(* CODESYS project TP2_INF_IND_RENAN_JULIA.project

Project tree, tasks and I/O mapping:
  Device : CODESYS Control Win V3, 3S - Smart Software Solutions GmbH, order no. 305021, version 3.5.11.40
    application Application
      libraries: Standard, * (System)
      task MainTask (cyclic, interval t#20ms, priority 1) calls Main
      task Simulacao (cyclic, interval t#20ms, priority 1) calls SimulacaoProcesso
      program Main [ST]
      Symbols
      function block AlarmLogic [ST]
      program SimulacaoProcesso [ST]
*)

// Device/Application/Main
PROGRAM Main
VAR_INPUT
    CMD_INICIAR_CARREGAMENTO: BOOL;
    CMD_INICIAR_DESCARREGAMENTO: BOOL;
    CAMINHAO_POSICIONADO: BOOL;
    CAPACIDADE_CAMINHAO: REAL;
    PESO_SILO1: REAL;
    PESO_SILO2: REAL;
    Modo_Automatico_Carregamento: BOOL;
    Modo_Automatico_Descarregamento: BOOL;
    CMD_MANUAL_VENTILACAO_SILO1: BOOL;
    CMD_MANUAL_VENTILACAO_SILO2: BOOL;
    CMD_MANUAL_ALIMENTADOR_MOEGA1_ON: BOOL;
    CMD_MANUAL_ALIMENTADOR_MOEGA2_ON: BOOL;
    CMD_MANUAL_TRANSPORTADOR_ENTRADA_ON: BOOL;
    CMD_MANUAL_TRANSPORTADOR_SAIDA_ON: BOOL;
    CMD_MANUAL_MOEGA_PESAGEM_ON: BOOL;
    CMD_MANUAL_ALIMENTADOR_SAIDA_ON: BOOL;
    CMD_MANUAL_DESVIADOR_MANGUEIRA: INT;
END_VAR

VAR_OUTPUT
    VENTILACAO_SILO1: BOOL := FALSE;
    VENTILACAO_SILO2: BOOL := FALSE;
    ALIMENTADOR_MOEGA1_ON: BOOL := FALSE;
    ALIMENTADOR_MOEGA2_ON: BOOL := FALSE;
    TRANSPORTADOR_SAIDA_ON: BOOL := FALSE;
    MOEGA_PESAGEM_ON: BOOL := FALSE;
    TRANSPORTADOR_ENTRADA_ON: BOOL := FALSE;
    DESVIADOR_MANGUEIRA: INT :=1;
END_VAR

VAR
	alarmLogic: AlarmLogic;
    NIVEL_BAIXO_SILO1: BOOL;
    NIVEL_BAIXO_SILO2: BOOL;
    NIVEL_ALTO_SILO1: BOOL;
    NIVEL_ALTO_SILO2: BOOL;
    PESO_MOEGA: REAL;
    TaxaTransferenciaCarregamento: REAL := 50.0;
    TaxaTransferenciaDescarregamento: REAL := 100.0;
    ALARME_CARREGAMENTO: BOOL;
    ALARME_DESCARREGAMENTO: BOOL;
    INICIAR_CARREGAMENTO: BOOL;
    INICIAR_DESCARREGAMENTO: BOOL;
    inicio_carregamento: TIME;
    inicio_descarregamento: TIME;
    SiloSelecionado: INT;
    VAGAO_POSICIONADO: BOOL;
    CAPACIDADE_VAGAO: REAL := 1000.0;
    VAGAO_CAPACIDADE_RESTANTE: REAL := 0.0;
    VAGAO_POSICIONADO_ANTERIOR: BOOL := FALSE;
    lastUpdateTime: TIME;
    elapsedTime: REAL;
    CAMINHAO_CHEIO: BOOL;
    equipmentOffTime: TIME;
    VAGAO_CHEIO: BOOL;
    CapacidadeDisponivelSilo1: REAL;
    CapacidadeDisponivelSilo2: REAL;
    CapacidadeTotalDisponivel: REAL;
    CapacidadeDescarregamento: REAL := 1000.0;
    CAMINHAO_POSICIONADO_ANTERIOR: BOOL := FALSE;
	ALARME_TRANSPORTADOR_ENTRADA_VAZIO: BOOL;
	ALARME_ALIMENTADOR_MOEGA_VAZIO: BOOL;
	ALARME_MOEGA_PESAGEM: BOOL;
	ALIMENTADOR_SAIDA_ON: BOOL;
	ALARME_TRANSPORTADOR_SAIDA_VAZIO: BOOL;
	ALARME_ALIMENTADOR_SAIDA: BOOL;
	ALARME_TRANSPORTADOR_SAIDA_ALIMENTADOR: BOOL;
	TRANSPORTADOR_ENTRADA_VAZIO_TIMER: TIME;
    TRANSPORTADOR_ENTRADA_VAZIO: BOOL := FALSE;
    
    PESO_TRANSPORTADOR_ENTRADA: REAL;
	ALARME_TRANSPORTADOR_ENTRADA_CHEIO: BOOL;
	TIMER_ALIMENTADOR_MOEGA1_VAZIO: TIME;
    ALARME_ALIMENTADOR_MOEGA1_VAZIO: BOOL := FALSE;
    ALARME_ALIMENTADOR_MOEGA1_CHEIO: BOOL := FALSE;
    PESO_ALIMENTADOR_MOEGA1: REAL; 

    TIMER_ALIMENTADOR_MOEGA2_VAZIO: TIME;
    ALARME_ALIMENTADOR_MOEGA2_VAZIO: BOOL := FALSE;
    ALARME_ALIMENTADOR_MOEGA2_CHEIO: BOOL := FALSE;
    PESO_ALIMENTADOR_MOEGA2: REAL;
	TIMER_TRANSPORTADOR_SAIDA_VAZIO: TIME;
	TIMER_TRANSPORTADOR_ENTRADA_VAZIO: TIME;
	PermiteMudancaModoCarregamento: BOOL := FALSE;
	PermiteMudancaModoDescarregamento: BOOL:= FALSE;
	VAGAO_FORA: BOOL;
	AUTORIZA_CARREGAMENTO: BOOL;
	ALARMES_DESLIGADOS: BOOL;
	DESCARREGAMENTO_EM_ANDAMENTO: BOOL;
END_VAR

alarmLogic.CURRENT_TIME := TIME();

// Configurar entradas do Function Block
alarmLogic.MOEGA_PESAGEM_ON := MOEGA_PESAGEM_ON;
alarmLogic.PESO_MOEGA := PESO_MOEGA;
alarmLogic.TRANSPORTADOR_SAIDA_ON := TRANSPORTADOR_SAIDA_ON;
alarmLogic.ALIMENTADOR_SAIDA_ON := ALIMENTADOR_SAIDA_ON;
alarmLogic.TRANSPORTADOR_ENTRADA_ON := TRANSPORTADOR_ENTRADA_ON;
alarmLogic.PESO_TRANSPORTADOR_ENTRADA := PESO_TRANSPORTADOR_ENTRADA;
alarmLogic.ALIMENTADOR_MOEGA1_ON := ALIMENTADOR_MOEGA1_ON;
alarmLogic.PESO_ALIMENTADOR_MOEGA1 := PESO_ALIMENTADOR_MOEGA1;
alarmLogic.ALIMENTADOR_MOEGA2_ON := ALIMENTADOR_MOEGA2_ON;
alarmLogic.PESO_ALIMENTADOR_MOEGA2 := PESO_ALIMENTADOR_MOEGA2;
alarmLogic.CAMINHAO_POSICIONADO := CAMINHAO_POSICIONADO;

// Chamar o Function Block
alarmLogic();

// Ler saídas do Function Block
ALARME_MOEGA_PESAGEM := alarmLogic.ALARME_MOEGA_PESAGEM;
ALARME_TRANSPORTADOR_SAIDA_VAZIO := alarmLogic.ALARME_TRANSPORTADOR_SAIDA_VAZIO;
ALARME_TRANSPORTADOR_SAIDA_ALIMENTADOR := alarmLogic.ALARME_TRANSPORTADOR_SAIDA_ALIMENTADOR;
ALARME_TRANSPORTADOR_ENTRADA_VAZIO := alarmLogic.ALARME_TRANSPORTADOR_ENTRADA_VAZIO;
ALARME_TRANSPORTADOR_ENTRADA_CHEIO := alarmLogic.ALARME_TRANSPORTADOR_ENTRADA_CHEIO;
ALARME_ALIMENTADOR_MOEGA1_VAZIO := alarmLogic.ALARME_ALIMENTADOR_MOEGA1_VAZIO;
ALARME_ALIMENTADOR_MOEGA1_CHEIO := alarmLogic.ALARME_ALIMENTADOR_MOEGA1_CHEIO;
ALARME_ALIMENTADOR_MOEGA2_VAZIO := alarmLogic.ALARME_ALIMENTADOR_MOEGA2_VAZIO;
ALARME_ALIMENTADOR_MOEGA2_CHEIO := alarmLogic.ALARME_ALIMENTADOR_MOEGA2_CHEIO;
ALARME_ALIMENTADOR_SAIDA := alarmLogic.ALARME_ALIMENTADOR_SAIDA;
ALARMES_DESLIGADOS    := alarmLogic.ALARMES_DESLIGADOS;

IF PESO_SILO1 <= 100 THEN
    NIVEL_BAIXO_SILO1 := TRUE;
ELSE
    NIVEL_BAIXO_SILO1 := FALSE;    
END_IF

IF PESO_SILO2 <= 100 THEN
    NIVEL_BAIXO_SILO2 := TRUE;
ELSE
    NIVEL_BAIXO_SILO2 := FALSE;    
END_IF

IF PESO_SILO1 >= 2400 THEN
    NIVEL_ALTO_SILO1 := TRUE;
ELSE
    NIVEL_ALTO_SILO1 := FALSE;    
END_IF

IF PESO_SILO2 >= 2400 THEN
    NIVEL_ALTO_SILO2 := TRUE;
ELSE 
    NIVEL_ALTO_SILO2 := FALSE;    
END_IF

IF TRANSPORTADOR_ENTRADA_ON AND (NOT VAGAO_POSICIONADO) THEN
	VAGAO_FORA := TRUE;
ELSE
    VAGAO_FORA := FALSE;	
END_IF

elapsedTime := TIME_TO_REAL(TIME() - lastUpdateTime) / 1000.0;
lastUpdateTime := TIME();

IF VAGAO_POSICIONADO AND NOT VAGAO_POSICIONADO_ANTERIOR THEN
    VAGAO_CAPACIDADE_RESTANTE := CAPACIDADE_VAGAO;
    VAGAO_POSICIONADO_ANTERIOR := TRUE;
    VAGAO_CHEIO := FALSE;
ELSIF NOT VAGAO_POSICIONADO THEN
    VAGAO_POSICIONADO_ANTERIOR := FALSE;
END_IF

IF CAMINHAO_POSICIONADO AND NOT CAMINHAO_POSICIONADO_ANTERIOR THEN
    CAMINHAO_POSICIONADO_ANTERIOR := TRUE;
    CAMINHAO_CHEIO := FALSE;
    AUTORIZA_CARREGAMENTO := TRUE; // Autoriza carregamento quando caminhão é reposicionado
ELSIF NOT CAMINHAO_POSICIONADO THEN
    CAMINHAO_POSICIONADO_ANTERIOR := FALSE;
    AUTORIZA_CARREGAMENTO := FALSE; // Reseta a autorização quando caminhão não está mais posicionado
END_IF

// Carregamento
IF Modo_Automatico_Carregamento THEN
    IF NOT INICIAR_CARREGAMENTO AND CMD_INICIAR_CARREGAMENTO AND AUTORIZA_CARREGAMENTO THEN
        IF CAMINHAO_POSICIONADO AND (CAPACIDADE_CAMINHAO >= 200 AND CAPACIDADE_CAMINHAO <= 800 AND (REAL_TO_INT(CAPACIDADE_CAMINHAO) MOD 50 = 0)) THEN
            IF ((PESO_SILO1 - 100) + (PESO_SILO2 - 100) >= CAPACIDADE_CAMINHAO) AND (NOT CAMINHAO_CHEIO) THEN
                INICIAR_CARREGAMENTO := TRUE;
                inicio_carregamento := TIME();
                ALARME_CARREGAMENTO := FALSE;

                IF PESO_SILO1 >= PESO_SILO2 THEN
                    SiloSelecionado := 1;
                ELSE
                    SiloSelecionado := 2;
                END_IF;
            ELSE
                ALARME_CARREGAMENTO := TRUE;
            END_IF
        ELSE
            ALARME_CARREGAMENTO := TRUE;
        END_IF
    END_IF

    IF INICIAR_CARREGAMENTO THEN
        IF (PESO_SILO1 >= 100 OR PESO_SILO2 >= 100) THEN
            TRANSPORTADOR_SAIDA_ON := TRUE;
            MOEGA_PESAGEM_ON := TRUE;
            ALIMENTADOR_SAIDA_ON := TRUE;

            IF PESO_MOEGA < CAPACIDADE_CAMINHAO THEN
                PESO_MOEGA := PESO_MOEGA + TaxaTransferenciaCarregamento * elapsedTime;
                IF SiloSelecionado = 1 THEN
                    IF NOT NIVEL_BAIXO_SILO1 THEN
                        VENTILACAO_SILO1 := TRUE; 
                        PESO_SILO1 := PESO_SILO1 - TaxaTransferenciaCarregamento * elapsedTime;
                        ALIMENTADOR_MOEGA1_ON := TRUE;
                        PESO_ALIMENTADOR_MOEGA1 := 1;
                        PESO_ALIMENTADOR_MOEGA2 := 0;
                        VENTILACAO_SILO2 := FALSE;
                        ALIMENTADOR_MOEGA2_ON := FALSE;
                    ELSE
                        SiloSelecionado := 2;
                        VENTILACAO_SILO1 := FALSE;
                        VENTILACAO_SILO2 := TRUE;
                    END_IF;
                ELSIF SiloSelecionado = 2 THEN
                    IF NOT NIVEL_BAIXO_SILO2 THEN
                        VENTILACAO_SILO2 := TRUE;
                        PESO_SILO2 := PESO_SILO2 - TaxaTransferenciaCarregamento * elapsedTime;
                        ALIMENTADOR_MOEGA2_ON := TRUE;
                        PESO_ALIMENTADOR_MOEGA1 := 0;
                        PESO_ALIMENTADOR_MOEGA2 := 1;
                        VENTILACAO_SILO1 := FALSE;
                        ALIMENTADOR_MOEGA1_ON := FALSE;
                    ELSE
                        SiloSelecionado := 1;
                        VENTILACAO_SILO1 := TRUE;
                        VENTILACAO_SILO2 := FALSE;
                    END_IF;
                END_IF;
            END_IF
        ELSE
            ALARME_CARREGAMENTO := TRUE;
            INICIAR_CARREGAMENTO := FALSE;
        END_IF;

        IF PESO_MOEGA >= CAPACIDADE_CAMINHAO OR ALARME_ALIMENTADOR_SAIDA THEN
            CAMINHAO_CHEIO := TRUE;
            INICIAR_CARREGAMENTO := FALSE;
            equipmentOffTime := TIME();
            AUTORIZA_CARREGAMENTO := FALSE; // Reseta a autorização após o carregamento ser concluído
        END_IF
    END_IF

    IF CAMINHAO_CHEIO THEN
        ALIMENTADOR_MOEGA1_ON := FALSE;
        PESO_ALIMENTADOR_MOEGA1 := 0;
        ALIMENTADOR_MOEGA2_ON := FALSE;
        PESO_ALIMENTADOR_MOEGA2 := 0;
        IF (TIME() - equipmentOffTime >= T#1S) THEN
            MOEGA_PESAGEM_ON := FALSE;
            PESO_MOEGA := 0;
        END_IF
        IF (TIME() - equipmentOffTime >= T#2S) THEN
            TRANSPORTADOR_SAIDA_ON := FALSE;
        END_IF
        IF (TIME() - equipmentOffTime >= T#3S) THEN
            ALIMENTADOR_SAIDA_ON := FALSE;
        END_IF
        IF (TIME() - equipmentOffTime >= T#5S) THEN
            VENTILACAO_SILO1 := FALSE;
            VENTILACAO_SILO2 := FALSE;
            CAMINHAO_CHEIO := FALSE;
        END_IF
    END_IF
END_IF

// Descarregamento
IF Modo_Automatico_Descarregamento THEN
    CapacidadeDisponivelSilo1 := 2400.0 - PESO_SILO1;
    CapacidadeDisponivelSilo2 := 2400.0 - PESO_SILO2;
    CapacidadeTotalDisponivel := CapacidadeDisponivelSilo1 + CapacidadeDisponivelSilo2;

    IF NOT INICIAR_DESCARREGAMENTO AND CMD_INICIAR_DESCARREGAMENTO THEN
        IF VAGAO_POSICIONADO AND (CapacidadeTotalDisponivel >= CapacidadeDescarregamento) AND (NOT VAGAO_CHEIO OR NOT VAGAO_FORA) AND NOT (NIVEL_ALTO_SILO1 AND NIVEL_ALTO_SILO2) THEN
            IF NOT ALARME_DESCARREGAMENTO THEN
                INICIAR_DESCARREGAMENTO := TRUE;
                inicio_descarregamento := TIME();
                ALARME_DESCARREGAMENTO := FALSE;

                IF (PESO_SILO1 < PESO_SILO2) AND (NOT NIVEL_ALTO_SILO1) THEN
                    DESVIADOR_MANGUEIRA := 1;
                    VENTILACAO_SILO1 := TRUE;
                    VENTILACAO_SILO2 := FALSE;
                ELSIF (PESO_SILO2 < PESO_SILO1) AND (NOT NIVEL_ALTO_SILO2) THEN
                    DESVIADOR_MANGUEIRA := 2;
                    VENTILACAO_SILO2 := TRUE;
                    VENTILACAO_SILO1 := FALSE;
                ELSIF (PESO_SILO1 = PESO_SILO2) THEN
                    IF NOT INICIAR_DESCARREGAMENTO THEN
                        IF DESVIADOR_MANGUEIRA = 1 THEN
                            SiloSelecionado := 1;
                            DESVIADOR_MANGUEIRA := 1;
                            VENTILACAO_SILO1 := TRUE;
                            VENTILACAO_SILO2 := FALSE;
                        ELSE
                            SiloSelecionado := 2;
                            DESVIADOR_MANGUEIRA := 2;
                            VENTILACAO_SILO2 := TRUE;
                            VENTILACAO_SILO1 := FALSE;
                        END_IF
                    END_IF
                END_IF
            END_IF
        ELSE
            ALARME_DESCARREGAMENTO := TRUE;
        END_IF
    END_IF

    IF INICIAR_DESCARREGAMENTO THEN
        TRANSPORTADOR_ENTRADA_ON := TRUE;
        
        PESO_TRANSPORTADOR_ENTRADA := 1;
        IF VAGAO_CAPACIDADE_RESTANTE > 0 THEN
            IF (NOT NIVEL_ALTO_SILO1) AND (DESVIADOR_MANGUEIRA = 1) THEN
                PESO_SILO1 := PESO_SILO1 + TaxaTransferenciaDescarregamento * elapsedTime;
                VAGAO_CAPACIDADE_RESTANTE := VAGAO_CAPACIDADE_RESTANTE - TaxaTransferenciaDescarregamento * elapsedTime;
                VENTILACAO_SILO1 := TRUE;
                VENTILACAO_SILO2 := FALSE;
                IF NIVEL_ALTO_SILO1 THEN
                    DESVIADOR_MANGUEIRA := 2;
                    VENTILACAO_SILO1 := FALSE;
                    VENTILACAO_SILO2 := TRUE;
                END_IF
            ELSE
                IF (NOT NIVEL_ALTO_SILO2) THEN
                    PESO_SILO2 := PESO_SILO2 + TaxaTransferenciaDescarregamento * elapsedTime;
                    VAGAO_CAPACIDADE_RESTANTE := VAGAO_CAPACIDADE_RESTANTE - TaxaTransferenciaDescarregamento * elapsedTime;
                    VENTILACAO_SILO2 := TRUE;
                    VENTILACAO_SILO1 := FALSE;
                    DESVIADOR_MANGUEIRA := 2;
                    
                END_IF
                IF NIVEL_ALTO_SILO2 THEN
                    DESVIADOR_MANGUEIRA := 1;
                    VENTILACAO_SILO2 := FALSE;
                    VENTILACAO_SILO1 := TRUE;
                END_IF
            END_IF

            IF VAGAO_CAPACIDADE_RESTANTE <= 0 OR VAGAO_FORA THEN
                VAGAO_CHEIO := TRUE;
                INICIAR_DESCARREGAMENTO := FALSE;
                equipmentOffTime := TIME();
            END_IF
        END_IF
    END_IF

    IF VAGAO_CHEIO THEN
        IF (TIME() - equipmentOffTime >= T#2S) THEN
            TRANSPORTADOR_ENTRADA_ON := FALSE;
            PESO_TRANSPORTADOR_ENTRADA := 0;
        END_IF
        IF (TIME() - equipmentOffTime >= T#5S) THEN
            VENTILACAO_SILO1 := FALSE;
            VENTILACAO_SILO2 := FALSE;
        END_IF
    END_IF

    // Redefinir alarme quando houver capacidade
    IF CapacidadeTotalDisponivel >= CapacidadeDescarregamento THEN
        ALARME_DESCARREGAMENTO := FALSE;
    END_IF
END_IF


IF NOT Modo_Automatico_Carregamento THEN
    IF ALARMES_DESLIGADOS THEN
        VENTILACAO_SILO1 := CMD_MANUAL_VENTILACAO_SILO1;
        VENTILACAO_SILO2 := CMD_MANUAL_VENTILACAO_SILO2;
        ALIMENTADOR_MOEGA1_ON := CMD_MANUAL_ALIMENTADOR_MOEGA1_ON;
        ALIMENTADOR_MOEGA2_ON := CMD_MANUAL_ALIMENTADOR_MOEGA2_ON;
        TRANSPORTADOR_SAIDA_ON := CMD_MANUAL_TRANSPORTADOR_SAIDA_ON;
        MOEGA_PESAGEM_ON := CMD_MANUAL_MOEGA_PESAGEM_ON;
    END_IF
END_IF

IF NOT Modo_Automatico_Descarregamento THEN
    IF ALARMES_DESLIGADOS THEN
        VENTILACAO_SILO1 := CMD_MANUAL_VENTILACAO_SILO1;
        VENTILACAO_SILO2 := CMD_MANUAL_VENTILACAO_SILO2;
        DESVIADOR_MANGUEIRA := CMD_MANUAL_DESVIADOR_MANGUEIRA;
        TRANSPORTADOR_ENTRADA_ON := CMD_MANUAL_TRANSPORTADOR_ENTRADA_ON;
    END_IF
END_IF

END_PROGRAM

// Device/Application/AlarmLogic
FUNCTION_BLOCK AlarmLogic
VAR_INPUT
    MOEGA_PESAGEM_ON: BOOL;
    PESO_MOEGA: REAL;
    TRANSPORTADOR_SAIDA_ON: BOOL;
    ALIMENTADOR_SAIDA_ON: BOOL;
    TRANSPORTADOR_ENTRADA_ON: BOOL;
    PESO_TRANSPORTADOR_ENTRADA: REAL;
    ALIMENTADOR_MOEGA1_ON: BOOL;
    PESO_ALIMENTADOR_MOEGA1: REAL;
    ALIMENTADOR_MOEGA2_ON: BOOL;
    PESO_ALIMENTADOR_MOEGA2: REAL;
	CURRENT_TIME: TIME;
	CAMINHAO_POSICIONADO :BOOL;
END_VAR

VAR_OUTPUT
    ALARME_MOEGA_PESAGEM: BOOL;
    ALARME_TRANSPORTADOR_SAIDA_VAZIO: BOOL;
    ALARME_TRANSPORTADOR_SAIDA_ALIMENTADOR: BOOL;
    ALARME_TRANSPORTADOR_ENTRADA_VAZIO: BOOL;
    ALARME_TRANSPORTADOR_ENTRADA_CHEIO: BOOL;
    ALARME_ALIMENTADOR_MOEGA1_VAZIO: BOOL;
    ALARME_ALIMENTADOR_MOEGA1_CHEIO: BOOL;
    ALARME_ALIMENTADOR_MOEGA2_VAZIO: BOOL;
    ALARME_ALIMENTADOR_MOEGA2_CHEIO: BOOL;
	ALARME_ALIMENTADOR_SAIDA : BOOL;
	ALARMES_DESLIGADOS: BOOL;
END_VAR

VAR
    TIMER_TRANSPORTADOR_SAIDA_VAZIO: TIME;
    TIMER_TRANSPORTADOR_ENTRADA_VAZIO: TIME;
    TIMER_ALIMENTADOR_MOEGA1_VAZIO: TIME;
    TIMER_ALIMENTADOR_MOEGA2_VAZIO: TIME;

	
END_VAR

// Alarme para moega de pesagem com peso diferente de zero e transportador de saída desligado
IF (MOEGA_PESAGEM_ON AND (PESO_MOEGA > 0)) AND NOT TRANSPORTADOR_SAIDA_ON THEN
    ALARME_MOEGA_PESAGEM := TRUE;
ELSE
    ALARME_MOEGA_PESAGEM := FALSE;
END_IF

// Alarme para transportador de saída vazio por mais de 5 segundos
IF TRANSPORTADOR_SAIDA_ON AND (PESO_MOEGA <= 0) THEN
    IF (CURRENT_TIME - TIMER_TRANSPORTADOR_SAIDA_VAZIO >= T#5S) THEN
        ALARME_TRANSPORTADOR_SAIDA_VAZIO := TRUE;
    END_IF
ELSE
    ALARME_TRANSPORTADOR_SAIDA_VAZIO := FALSE;
    TIMER_TRANSPORTADOR_SAIDA_VAZIO := CURRENT_TIME;
END_IF

// Alarme para transportador de saída ligado e alimentador de saída desligado
IF TRANSPORTADOR_SAIDA_ON AND NOT ALIMENTADOR_SAIDA_ON THEN
    ALARME_TRANSPORTADOR_SAIDA_ALIMENTADOR := TRUE;
ELSE
    ALARME_TRANSPORTADOR_SAIDA_ALIMENTADOR := FALSE;
END_IF

// Alarme para transportador de entrada vazio por mais de 5 segundos
IF TRANSPORTADOR_ENTRADA_ON AND (PESO_TRANSPORTADOR_ENTRADA <= 0) THEN
    IF (CURRENT_TIME - TIMER_TRANSPORTADOR_ENTRADA_VAZIO >= T#5S) THEN
        ALARME_TRANSPORTADOR_ENTRADA_VAZIO := TRUE;
    END_IF
ELSE
    ALARME_TRANSPORTADOR_ENTRADA_VAZIO := FALSE;
    TIMER_TRANSPORTADOR_ENTRADA_VAZIO := CURRENT_TIME;
END_IF

// Alarme para transportador de entrada quando há material dentro de si
IF TRANSPORTADOR_ENTRADA_ON AND (PESO_TRANSPORTADOR_ENTRADA > 0) THEN
    ALARME_TRANSPORTADOR_ENTRADA_CHEIO := TRUE;
ELSE
    ALARME_TRANSPORTADOR_ENTRADA_CHEIO := FALSE;
END_IF

// Alarme para Alimentador da Moega 1 vazio por mais de 5 segundos
IF ALIMENTADOR_MOEGA1_ON AND (PESO_ALIMENTADOR_MOEGA1 <= 0) THEN
    IF (CURRENT_TIME - TIMER_ALIMENTADOR_MOEGA1_VAZIO >= T#5S) THEN
        ALARME_ALIMENTADOR_MOEGA1_VAZIO := TRUE;
    END_IF
ELSE
    ALARME_ALIMENTADOR_MOEGA1_VAZIO := FALSE;
    TIMER_ALIMENTADOR_MOEGA1_VAZIO := CURRENT_TIME;
END_IF

// Alarme para Alimentador da Moega 1 quando há grãos no alimentador
IF ALIMENTADOR_MOEGA1_ON AND (PESO_ALIMENTADOR_MOEGA1 > 0) THEN
    ALARME_ALIMENTADOR_MOEGA1_CHEIO := TRUE;
ELSE
    ALARME_ALIMENTADOR_MOEGA1_CHEIO := FALSE;
END_IF

// Alarme para Alimentador da Moega 2 vazio por mais de 5 segundos
IF ALIMENTADOR_MOEGA2_ON AND (PESO_ALIMENTADOR_MOEGA2 <= 0) THEN
    IF (CURRENT_TIME - TIMER_ALIMENTADOR_MOEGA2_VAZIO >= T#5S) THEN
        ALARME_ALIMENTADOR_MOEGA2_VAZIO := TRUE;
    END_IF
ELSE
    ALARME_ALIMENTADOR_MOEGA2_VAZIO := FALSE;
    TIMER_ALIMENTADOR_MOEGA2_VAZIO := CURRENT_TIME;
END_IF

// Alarme para Alimentador da Moega 2 quando há grãos no alimentador
IF ALIMENTADOR_MOEGA2_ON AND (PESO_ALIMENTADOR_MOEGA2 > 0) THEN
    ALARME_ALIMENTADOR_MOEGA2_CHEIO := TRUE;
ELSE
    ALARME_ALIMENTADOR_MOEGA2_CHEIO := FALSE;
END_IF

IF ALIMENTADOR_SAIDA_ON AND (NOT CAMINHAO_POSICIONADO) THEN
	ALARME_ALIMENTADOR_SAIDA := TRUE;
ELSE
    ALARME_ALIMENTADOR_SAIDA := FALSE;	
END_IF


IF NOT ALARME_ALIMENTADOR_SAIDA AND (NOT ALARME_ALIMENTADOR_MOEGA2_CHEIO) AND (NOT ALARME_ALIMENTADOR_MOEGA2_VAZIO) AND (NOT ALARME_ALIMENTADOR_MOEGA1_CHEIO) AND (NOT ALARME_ALIMENTADOR_MOEGA1_VAZIO) 
     AND (NOT ALARME_TRANSPORTADOR_ENTRADA_CHEIO) AND(NOT ALARME_TRANSPORTADOR_ENTRADA_VAZIO) AND (NOT ALARME_TRANSPORTADOR_SAIDA_ALIMENTADOR) AND (NOT ALARME_TRANSPORTADOR_SAIDA_VAZIO) THEN
      ALARMES_DESLIGADOS := TRUE;
END_IF

END_FUNCTION_BLOCK

// Device/Application/SimulacaoProcesso
PROGRAM SimulacaoProcesso
VAR_INPUT
    TRANSPORTADOR_ENTRADA_ON: BOOL;
    TRANSPORTADOR_SAIDA_ON: BOOL;
    VENTILACAO_SILO1: BOOL;
    VENTILACAO_SILO2: BOOL;
    ALIMENTADOR_MOEGA1_ON: BOOL;
    ALIMENTADOR_MOEGA2_ON: BOOL;
    CAMINHAO_POSICIONADO: BOOL;
    VAGAO_POSICIONADO: BOOL;
END_VAR

VAR_OUTPUT
    PESO_SILO1: REAL;
    PESO_SILO2: REAL;
    PESO_MOEGA: REAL;
    SENSOR_GRAO_ALIMENTADOR_MOEGA1: BOOL;
    SENSOR_GRAO_ALIMENTADOR_MOEGA2: BOOL;
    NIVEL_ALTO_SILO1: BOOL;
    NIVEL_ALTO_SILO2: BOOL;
    NIVEL_BAIXO_SILO1: BOOL;
    NIVEL_BAIXO_SILO2: BOOL;
    PESO_TRANSPORTADOR_ENTRADA: REAL;
    PESO_TRANSPORTADOR_SAIDA: REAL;
END_VAR

VAR
    taxa_transferencia_entrada: REAL := 100.0; // Taxa de transferência do transportador de entrada (kg/s)
    taxa_transferencia_saida: REAL := 50.0; // Taxa de transferência do transportador de saída (kg/s)
    tempo_atual: TIME;
    tempo_anterior: TIME := T#0s;
    delta_t: REAL;
END_VAR

// Calcular delta_t
tempo_atual := TIME();
delta_t := TIME_TO_REAL(tempo_atual - tempo_anterior) / 1000.0; // Converter TIME para segundos

// Inicializar variáveis de saída
PESO_TRANSPORTADOR_ENTRADA := 0.0;
PESO_TRANSPORTADOR_SAIDA := 0.0;

// Simular o comportamento dos silos e transportadores
IF TRANSPORTADOR_ENTRADA_ON THEN
    PESO_TRANSPORTADOR_ENTRADA := taxa_transferencia_entrada * delta_t;
    IF VAGAO_POSICIONADO THEN
        IF ALIMENTADOR_MOEGA1_ON THEN
            PESO_SILO1 := PESO_SILO1 + PESO_TRANSPORTADOR_ENTRADA;
            PESO_MOEGA := PESO_MOEGA - PESO_TRANSPORTADOR_ENTRADA;
        ELSIF ALIMENTADOR_MOEGA2_ON THEN
            PESO_SILO2 := PESO_SILO2 + PESO_TRANSPORTADOR_ENTRADA;
            PESO_MOEGA := PESO_MOEGA - PESO_TRANSPORTADOR_ENTRADA;
        END_IF
    END_IF
END_IF

IF TRANSPORTADOR_SAIDA_ON THEN
    PESO_TRANSPORTADOR_SAIDA := taxa_transferencia_saida * delta_t;
    IF CAMINHAO_POSICIONADO THEN
        IF ALIMENTADOR_MOEGA1_ON THEN
            PESO_MOEGA := PESO_MOEGA + PESO_TRANSPORTADOR_SAIDA;
            PESO_SILO1 := PESO_SILO1 - PESO_TRANSPORTADOR_SAIDA;
        ELSIF ALIMENTADOR_MOEGA2_ON THEN
            PESO_MOEGA := PESO_MOEGA + PESO_TRANSPORTADOR_SAIDA;
            PESO_SILO2 := PESO_SILO2 - PESO_TRANSPORTADOR_SAIDA;
        END_IF
    END_IF
END_IF

// Atualizar sensores de grãos
SENSOR_GRAO_ALIMENTADOR_MOEGA1 := (PESO_SILO1 > 0);
SENSOR_GRAO_ALIMENTADOR_MOEGA2 := (PESO_SILO2 > 0);

// Verificar níveis altos e baixos dos silos
NIVEL_ALTO_SILO1 := (PESO_SILO1 >= 2400);
NIVEL_ALTO_SILO2 := (PESO_SILO2 >= 2400);
NIVEL_BAIXO_SILO1 := (PESO_SILO1 <= 100);
NIVEL_BAIXO_SILO2 := (PESO_SILO2 <= 100);

// Atualizar o tempo anterior
tempo_anterior := tempo_atual;

END_PROGRAM
